# B&R Automation Studio project Lab_4
Automation Studio 4.5.2.102

## Configuration Config1

### Task classes (Cpu.sw)
```
Cyclic#1:
  Program <- Program.prg
VcDataObjects: Visu <- Visu.dob
Binaries: vcpfpp30, vcmgr, arsvcreg, arialbd, udbdef, vcpdsw, vcalarm, vccdt, vccbmp, vcgclass, Visu01, vctcal, vcshared, TCData, vccbtn, vcfile, Visu02, vcdsint, Visu03, vcrt, vcpfmtcx, vcbclass, vcfntttf, vcptelo, vcdsloc, vccovl, vcpdpp30, arial, Role, iomap, arconfig, asfw, sysconf, User, ashwac, ashwd
Libraries: McBase, runtime, fileio, vcresman, dataobj, Library
```

### IoMap.iom - 4PP065_0571_P74/IoMap.iom
```iecst
VAR_CONFIG
	::Program:real_motor_speed AT %IW."8I64xxxxxxx.00x-1".RFRD_Input;
	::Program:motor_speed AT %QW."8I64xxxxxxx.00x-1".LFRD_Output;
	::LED[0] AT %QX."X20DO9322".DigitalOutput02;
	::LED[1] AT %QX."X20DO9322".DigitalOutput03;
	::LED[2] AT %QX."X20DO9322".DigitalOutput04;
	::LED[3] AT %QX."X20DO9322".DigitalOutput05;
	::Program:servo.STATE  AT %IW."8I64xxxxxxx.00x-1".ETAD_Input;
	::Program:servo.COM  AT %QW."8I64xxxxxxx.00x-1".CMDD_Output;
END_VAR
```

## Logical view

Binary libraries used (declarations not repeated): Library

### Global.var - Global variables
```iecst
VAR
	LED : ARRAY[0..3] OF BOOL := [4(FALSE)];
	BTN : ARRAY[0..3] OF BOOL;
	blink : BOOL;
	motor_speed : INT := 0;
	real_motor_speed : INT;
END_VAR
```

### Program Logical/Program (ANSIC)

#### Variables.var
```iecst
VAR
	EVIRD : DRIVE;
	Counter : USINT;
END_VAR
```

#### Main.c
```c
#include <bur/plctypes.h>

#ifdef _DEFAULT_INCLUDES
#include <AsDefault.h>
#endif

void _INIT ProgramInit(void) {
}

void _CYCLIC ProgramCyclic(void) {
	DRIVE(&servo);

	if (blink) {
		if (Counter % 2) LED[0] = !LED[0];
		if (Counter % 5) LED[1] = !LED[1];
		if (Counter % 10) LED[2] = !LED[2];
		if (Counter % 20) LED[3] = !LED[3];
		Counter++;
	} else {
		int i;
		for (i = 0; i < 4; i++) LED[i] = BTN[i];
	}
}

void _EXIT ProgramExit(void) {

}
```

- Visualisation Logical/Visu (not shown)

Listed in the project but not available here: Logical/Global.typ, Logical/Libraries
